{attribute 'qualified_only'}
{attribute 'strict'}
TYPE machineStates :
(
	START_OF_DAY,
	DURING_DAY,
	END_OF_DAY,
	DISARMED
);
END_TYPE

(* stored: Version 1.1.0.1, ProductVersion 3.1.4024.12
   DUT machineStates: Id {b62a9363-bcb5-4c40-8785-1a67fe4adfd8} *)
